// TIA Portal V18 export
DATA_BLOCK "L1_TestiDS"   // DB29
{ S7_Optimized_Access := 'TRUE' }
VERSION : 0.1
// stored: AutoNumber false, DBAccessibleFromOPCUA true, DBAccessibleFromWebserver true, IsOnlyStoredInLoadMemory false, IsRetainMemResEnabled false, IsWriteProtectedInAS false, MemoryReserve 100
   VAR
      stz_selezionata : Int;
      stz : Array[1.."N_STAZIONI"] of Struct
         testo : Array[1.."N_DS"] of WString;
      END_STRUCT;
   END_VAR
BEGIN
END_DATA_BLOCK
